{region '#Template'}
	{attribute 'Version' := '5.0.0.0'}
	{attribute 'Tags' := '"LCID": "1031", "Text": "Fassade, Sonnenschutz, Parkposition"'}
	{attribute 'Tags' := '"LCID": "1033", "Text": "Facade, Sunprotection, parking position"'}
	{attribute 'Using' := '"Type": "Template", "URI": "ST_BA_SunBld"'}
	{attribute 'Using' := '"Type": "Template", "URI": "E_BA_SunBldPrio"'}
	{attribute 'Description' := '"LCID": "1031", "Text": "Sonnenschutz Parkposition"'}
	{attribute 'Description' := '"LCID": "1033", "Text": "Sunprotection parking-position"'}
{endregion}
FUNCTION_BLOCK FB_BA_Facade_ParkPosition EXTENDS FB_BA_View
VAR_INPUT
END_VAR
VAR_OUTPUT
	stSunBld					: ST_BA_SunBld;
	bParkPosEvent				: BOOL;	
END_VAR
VAR_INPUT CONSTANT
	FcdParkEn					: FB_BA_BV_Op;		
	FcdParkPos					: FB_BA_AV_Op;		
	FcdParkAngl					: FB_BA_AV_Op;		
	FcdParkPosEvent				: FB_BA_SunBldEvt :=(ePrio:=E_BA_SunBldPrio.eParkPosition);					
END_VAR
VAR
END_VAR

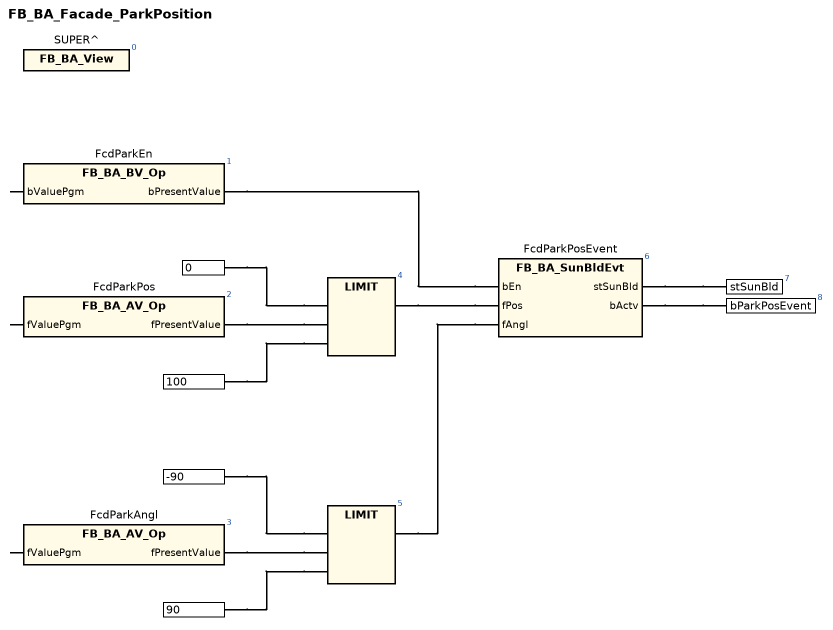
SUPER^(); // FB_BA_View
FcdParkEn(); // FB_BA_BV_Op
FcdParkPos(); // FB_BA_AV_Op
FcdParkAngl(); // FB_BA_AV_Op
FcdParkPosEvent(
    bEn := FcdParkEn.bPresentValue,
    fPos := LIMIT(0, FcdParkPos.fPresentValue, 100),
    fAngl := LIMIT(-90, FcdParkAngl.fPresentValue, 90)); // FB_BA_SunBldEvt
stSunBld := FcdParkPosEvent.stSunBld;
bParkPosEvent := FcdParkPosEvent.bActv;

METHOD FB_init : BOOL
VAR_INPUT
	bInitRetains : BOOL; // if TRUE; the retain variables are initialized (warm start / cold start)
	bInCopyCode : BOOL;  // if TRUE; the instance afterwards gets moved into the copy code (online change)
END_VAR
FcdParkEn.iParent				:= THIS^;
FcdParkEn.iLabel				:= LblCtl_FacadeParkingEnable;
FcdParkEn.sObjectName			:= '{Idx=01}';
FcdParkEn.sInactiveText			:= txtEvent_Off;
FcdParkEn.sActiveText			:= txtEvent_On;
FcdParkEn.bValueRm				:= FALSE;
FcdParkEn.eToggleMode			:= E_BA_ToggleMode.eSwitch;        

FcdParkPos.iParent				:= THIS^;
FcdParkPos.iLabel				:= LblCtl_FacadeParkingPosition;
FcdParkPos.sObjectName			:= '{Idx=01}';
FcdParkPos.eUnit				:= E_BA_Unit.eOther_Percent; 
FcdParkPos.fValueRm				:= 0.0;
FcdParkPos.fCOVIncrement		:= BA2_Param.fDefCOVIncrement;
		  
FcdParkAngl.iParent				:= THIS^;
FcdParkAngl.iLabel				:= LblCtl_FacadeParkingAngle;
FcdParkAngl.sObjectName			:= '{Idx=02}';
FcdParkAngl.eUnit				:= E_BA_Unit.eOther_DegreesAngular; 
FcdParkAngl.fValueRm			:= 0.0; 
FcdParkAngl.fCOVIncrement		:= BA2_Param.fDefCOVIncrement;
END_METHOD

END_FUNCTION_BLOCK

(* stored: Version 1.1.0.1, ProductVersion 3.1.4024.12
   POU FB_BA_Facade_ParkPosition: Id {be5fb990-fc5b-47e6-bf74-f8b5f5ea9d68}, SpecialFunc None
   Method FB_init: Id {25e0d6dd-262a-4a83-a14d-d25740876de1} *)
